// TIA Portal V20 export
TYPE "UDT_MTP_LockView8"
// Interface Definition LockView8
   STRUCT
      OSLevel : Byte := 16#00;   // OSLevel variable
      WQC { ExternalWritable := 'False'} : Byte := 16#FF;   // Worst Quality Code variable
      Logic { ExternalWritable := 'False'} : Bool;   // Logical behaviour, false: OR, true: AND
      In1En { ExternalWritable := 'False'} : Bool;   // Locking Input 1 - Enable, 0: Input not used, 1: Input is used
      In1 { ExternalWritable := 'False'} : Bool;   // Locking Input 1 - Value
      In1QC { ExternalWritable := 'False'} : Byte := 16#FF;   // Locking Input 1 - Quality Code
      In1Inv { ExternalWritable := 'False'} : Bool;   // Locking Input 1 - Inversion Enable, 0: Input not inverted, 1: Input inverted
      In1Txt { ExternalWritable := 'False'} : String[16] := '';   // Locking Input 1 - Additional Text
      In2En { ExternalWritable := 'False'} : Bool;   // Locking Input 2 - Enable, 0: Input not used, 1: Input is used
      In2 { ExternalWritable := 'False'} : Bool;   // Locking Input 2 - Value
      In2QC { ExternalWritable := 'False'} : Byte := 16#FF;   // Locking Input 2 - Quality Code
      In2Inv { ExternalWritable := 'False'} : Bool;   // Locking Input 2 - Inversion Enable, 0: Input not inverted, 1: Input inverted
      In2Txt { ExternalWritable := 'False'} : String[16] := '';   // Locking Input 2 - Additional Text
      In3En { ExternalWritable := 'False'} : Bool;   // Locking Input 3 - Enable, 0: Input not used, 1: Input is used
      In3 { ExternalWritable := 'False'} : Bool;   // Locking Input 3 - Value
      In3QC { ExternalWritable := 'False'} : Byte := 16#FF;   // Locking Input 3 - Quality Code
      In3Inv { ExternalWritable := 'False'} : Bool;   // Locking Input 3 - Inversion Enable, 0: Input not inverted, 1: Input inverted
      In3Txt { ExternalWritable := 'False'} : String[16] := '';   // Locking Input 3 - Additional Text
      In4En { ExternalWritable := 'False'} : Bool;   // Locking Input 4 - Enable, 0: Input not used, 1: Input is used
      In4 { ExternalWritable := 'False'} : Bool;   // Locking Input 4 - Value
      In4QC { ExternalWritable := 'False'} : Byte := 16#FF;   // Locking Input 4 - Quality Code
      In4Inv { ExternalWritable := 'False'} : Bool;   // Locking Input 4 - Inversion Enable, 0: Input not inverted, 1: Input inverted
      In4Txt { ExternalWritable := 'False'} : String[16] := '';   // Locking Input 4 - Additional Text
      In5En { ExternalWritable := 'False'} : Bool;   // Locking Input 5 - Enable, 0: Input not used, 1: Input is used
      In5 { ExternalWritable := 'False'} : Bool;   // Locking Input 5 - Value
      In5QC { ExternalWritable := 'False'} : Byte := 16#FF;   // Locking Input 5 - Quality Code
      In5Inv { ExternalWritable := 'False'} : Bool;   // Locking Input 5 - Inversion Enable, 0: Input not inverted, 1: Input inverted
      In5Txt { ExternalWritable := 'False'} : String[16] := '';   // Locking Input 5 - Additional Text
      In6En { ExternalWritable := 'False'} : Bool;   // Locking Input 6 - Enable, 0: Input not used, 1: Input is used
      In6 { ExternalWritable := 'False'} : Bool;   // Locking Input 6 - Value
      In6QC { ExternalWritable := 'False'} : Byte := 16#FF;   // Locking Input 6 - Quality Code
      In6Inv { ExternalWritable := 'False'} : Bool;   // Locking Input 6 - Inversion Enable, 0: Input not inverted, 1: Input inverted
      In6Txt { ExternalWritable := 'False'} : String[16] := '';   // Locking Input 6 - Additional Text
      In7En { ExternalWritable := 'False'} : Bool;   // Locking Input 7 - Enable, 0: Input not used, 1: Input is used
      In7 { ExternalWritable := 'False'} : Bool;   // Locking Input 7 - Value
      In7QC { ExternalWritable := 'False'} : Byte := 16#FF;   // Locking Input 7 - Quality Code
      In7Inv { ExternalWritable := 'False'} : Bool;   // Locking Input 7 - Inversion Enable, 0: Input not inverted, 1: Input inverted
      In7Txt { ExternalWritable := 'False'} : String[16] := '';   // Locking Input 7 - Additional Text
      In8En { ExternalWritable := 'False'} : Bool;   // Locking Input 8 - Enable, 0: Input not used, 1: Input is used
      In8 { ExternalWritable := 'False'} : Bool;   // Locking Input 8 - Value
      In8QC { ExternalWritable := 'False'} : Byte := 16#FF;   // Locking Input 8 - Quality Code
      In8Inv { ExternalWritable := 'False'} : Bool;   // Locking Input 8 - Inversion Enable, 0: Input not inverted, 1: Input inverted
      In8Txt { ExternalWritable := 'False'} : String[16] := '';   // Locking Input 8 - Additional Text
      Out { ExternalWritable := 'False'} : Bool;   // Locking Result Output
      OutQC { ExternalWritable := 'False'} : Byte := 16#FF;   // Locking Result Output - Quality Code
   END_STRUCT;
END_TYPE
